// TIA Portal V19 export
TYPE "lexchangetray_typeroller_signalTM_Simulation"
// Type: Bool
// stored: Access Published
   STRUCT
      trayAutomaticDischargeDetectionEm1 : Bool;
      trayAutomaticFeedingDetectionEm1 : Bool;
      restraintTrayAntiReverseDetection2Em1 : Bool;
      restraintTrayAntiReverseDetection1Em1 : Bool;
   END_STRUCT;
END_TYPE
